FUNCTION_BLOCK FB_FastFault
VAR_INPUT
	i_xReset		:	BOOL; //Set true to reset fast fault when errors are cleared
	i_xVetoBypass	:	BOOL; //Set true to bypass fast fault, connect to veto device
	
	i_xErrorInput		:	BOOL; //Set true to indicate error
END_VAR
VAR_OUTPUT
	q_xFastFaultOutput	:	BOOL;
END_VAR
VAR
	fbLatch	:	RS;
END_VAR
VAR // added by the converter: edge detectors and wires of the graphical bodies
    _ft1 : F_TRIG;
END_VAR

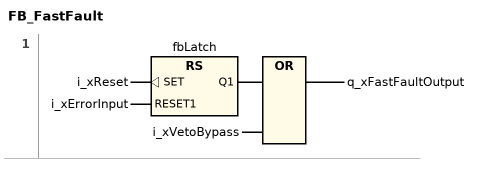
// NETWORK 1
_ft1(CLK := i_xReset);
fbLatch(SET := _ft1.Q, RESET1 := i_xErrorInput); // RS
q_xFastFaultOutput := fbLatch.Q1 OR i_xVetoBypass;

END_FUNCTION_BLOCK

(* stored: Version 1.1.0.1, ProductVersion 3.1.4020.12
   POU FB_FastFault: Id {40180f4a-e9df-0382-08a0-658ade013089}, SpecialFunc None *)
